{attribute 'GeneratedUsingTerminal: EP9224-0023-0016'}
{attribute addProperty BoxType "EP9224-0023-0016"}
{attribute addProperty Id "Temperature_WarningAT %I*BOOL1Temperature_ErrorAT %I*BOOL1Us_WarningAT %I*BOOL1Us_ErrorAT %I*BOOL1Up_WarningAT %I*BOOL1Up_ErrorAT %I*BOOL1Global_Error_BitAT %I*BOOL1Sum_Current_WarningAT %I*BOOL1Sum_Current_ErrorAT %I*BOOL1Reset_InputAT %I*BOOL1TxPDO_StateAT %I*BOOL1TxPDO_ToggleAT %I*BOOL1Current_UsAT %I*INT2Current_UpAT %I*INT2Voltage_UsAT %I*INT2Voltage_UpAT %I*INT2TemperatureAT %I*INT2"}
{attribute addProperty CRC "2569281258"}
{attribute addProperty Size "22"}
TYPE DPO_Inputs_Device_99241EEA :
STRUCT
	{attribute addProperty Name "Temperature_Warning"}
	Temperature_Warning AT %I* : BOOL;
	{attribute addProperty Name "Temperature_Error"}
	Temperature_Error AT %I* : BOOL;
	{attribute addProperty Name "Us_Warning"}
	Us_Warning AT %I* : BOOL;
	{attribute addProperty Name "Us_Error"}
	Us_Error AT %I* : BOOL;
	{attribute addProperty Name "Up_Warning"}
	Up_Warning AT %I* : BOOL;
	{attribute addProperty Name "Up_Error"}
	Up_Error AT %I* : BOOL;
	{attribute addProperty Name "Global_Error_Bit"}
	Global_Error_Bit AT %I* : BOOL;
	{attribute addProperty Name "Sum_Current_Warning"}
	Sum_Current_Warning AT %I* : BOOL;
	{attribute addProperty Name "Sum_Current_Error"}
	Sum_Current_Error AT %I* : BOOL;
	{attribute addProperty Name "Reset_Input"}
	Reset_Input AT %I* : BOOL;
	{attribute addProperty Name "TxPDO_State"}
	TxPDO_State AT %I* : BOOL;
	{attribute addProperty Name "TxPDO_Toggle"}
	TxPDO_Toggle AT %I* : BOOL;
	{attribute addProperty Name "Current_Us"}
	Current_Us AT %I* : INT;
	{attribute addProperty Name "Current_Up"}
	Current_Up AT %I* : INT;
	{attribute addProperty Name "Voltage_Us"}
	Voltage_Us AT %I* : INT;
	{attribute addProperty Name "Voltage_Up"}
	Voltage_Up AT %I* : INT;
	{attribute addProperty Name "Temperature"}
	Temperature AT %I* : INT;
END_STRUCT
END_TYPE

(* stored: Version 1.2.0.0, ProductVersion 3.1.4024.9
   DUT DPO_Inputs_Device_99241EEA: Id {5f839991-38b9-4f66-b466-26b9497f242f} *)
